FUNCTION_BLOCK X2Y2 (* Compute X^2-Y^2(event-driven) *)
  (* Standard: 61499-1 *)
  (* Version 0.1.1, 2006-02-16, JHC, Holobloc Inc, Testing new Save functions *)
  (* Version 0.0, 2001-10-08, JHC, Rockwell Automation *)
  (* Compiler header: package fb.rt.student; import fb.rt.math.*; *)
  (* Compiler Java Sun JDK 1.4.2 *)
  (* Compiler Java IBM Jikes 1.0.6 *)
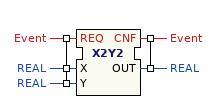
  EVENT_INPUT
    REQ WITH X, Y;
  END_EVENT
  EVENT_OUTPUT
    CNF WITH OUT;
  END_EVENT
  VAR_INPUT
    X : REAL;
    Y : REAL;
  END_VAR
  VAR_OUTPUT
    OUT : REAL;
  END_VAR
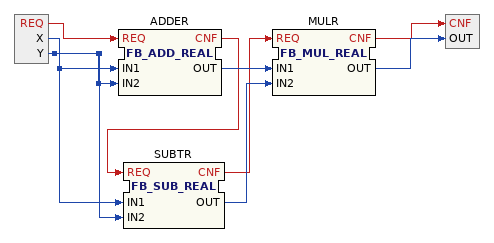
  FBS
    ADDER : FB_ADD_REAL;
    SUBTR : FB_SUB_REAL;
    MULR : FB_MUL_REAL;
  END_FBS
  EVENT_CONNECTIONS
    REQ TO ADDER.REQ;
    ADDER.CNF TO SUBTR.REQ;
    SUBTR.CNF TO MULR.REQ;
    MULR.CNF TO CNF;
  END_CONNECTIONS
  DATA_CONNECTIONS
    X TO ADDER.IN1;
    Y TO ADDER.IN2;
    X TO SUBTR.IN1;
    Y TO SUBTR.IN2;
    ADDER.OUT TO MULR.IN1;
    SUBTR.OUT TO MULR.IN2;
    MULR.OUT TO OUT;
  END_CONNECTIONS
END_FUNCTION_BLOCK
